TYPE ST_XtsCommandFeedback :
STRUCT
		(* Returns wether the execution of the method is done. *)
		IsDone : BOOL;
		(* Returns wether the execution of the method is busy. *)
		IsBusy : BOOL;
		(* Returns wether the execution of the method is busy. *)
		HasError : BOOL;
		(* Returns the HRESULT to the call. *)
		{attribute 'GUID' := '18071995-0000-0000-0000-000000000019'}
		{attribute 'GlobalType'}
		HRESULT : GLOBAL.HRESULT;
	END_STRUCT
END_TYPE

(* stored: Version 1.1.0.1, ProductVersion 3.1.4026.8
   DUT DUT: Id {de7bdfb9-08e8-4f12-99ca-b68db8892940} *)
